FUNCTION_BLOCK "GBK_TO_UNI"
{ S7_Optimized_Access := 'TRUE' }
VERSION : 0.1
   VAR_INPUT
      GBK : Word;
   END_VAR

   VAR_OUTPUT
      UNICODE : Word;
   END_VAR

   VAR
